// LS Electric XG5000 project: 신호등
// PLC LSPLC

PROGRAM NewProgram (task: 스캔 프로그램)

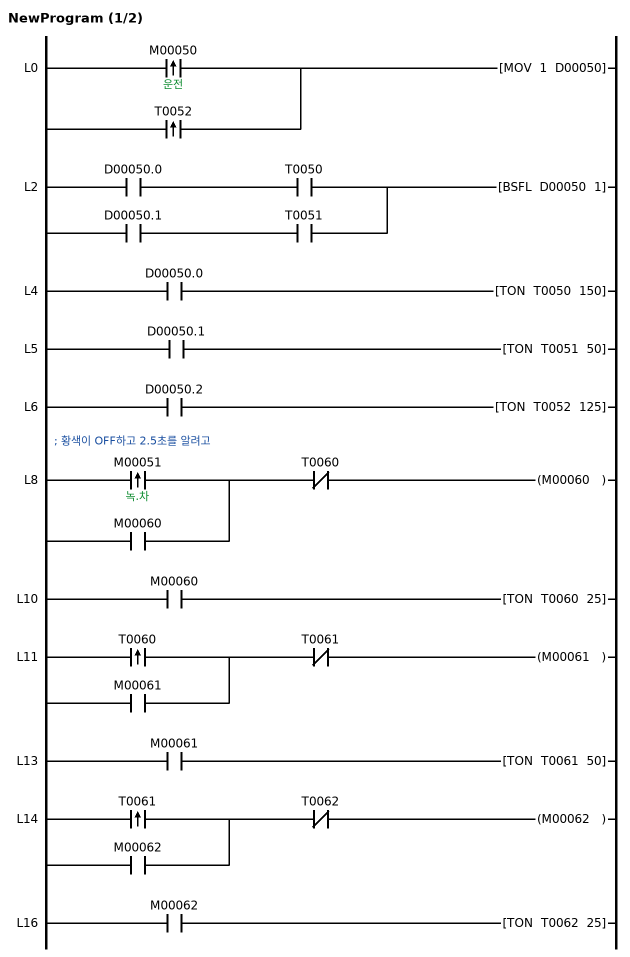
; L0
LOADP     M00050	// 운전
ORP       T0052
MOV       1 D00050
; L2
LOAD      D00050.0
AND       T0050
LOAD      D00050.1
AND       T0051
OR LOAD
BSFL      D00050 1
; L4
LOAD      D00050.0
TON       T0050 150
; L5
LOAD      D00050.1
TON       T0051 50
; L6
LOAD      D00050.2
TON       T0052 125
// 황색이 OFF하고 2.5초를 알려고
; L8
LOADP     M00051	// 녹.차
OR        M00060
AND NOT   T0060
OUT       M00060
; L10
LOAD      M00060
TON       T0060 25
; L11
LOADP     T0060
OR        M00061
AND NOT   T0061
OUT       M00061
; L13
LOAD      M00061
TON       T0061 50
; L14
LOADP     T0061
OR        M00062
AND NOT   T0062
OUT       M00062
; L16
LOAD      M00062
TON       T0062 25

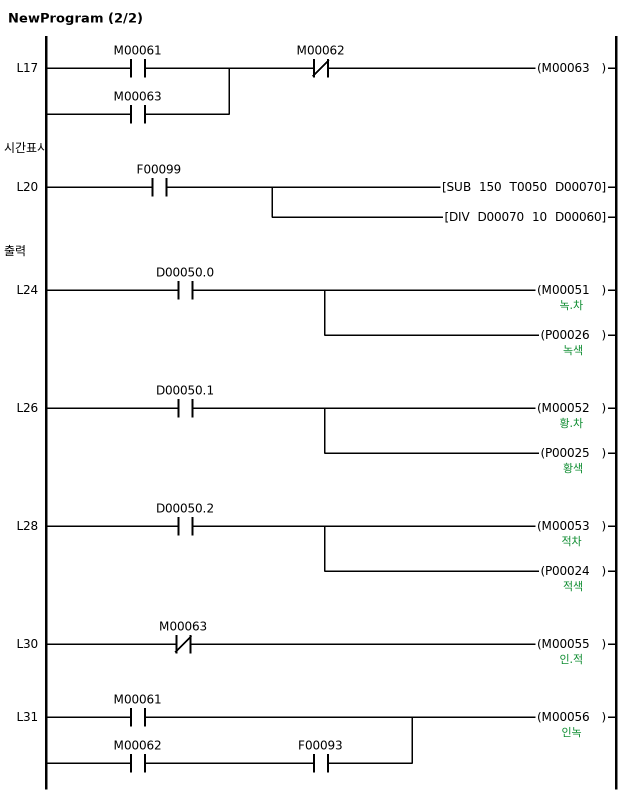
; L17
LOAD      M00061
OR        M00063
AND NOT   M00062
OUT       M00063
시간표시:
; L20
LOAD      F00099
SUB       150 T0050 D00070
DIV       D00070 10 D00060
출력:
; L24
LOAD      D00050.0
OUT       M00051	// 녹.차
OUT       P00026	// 녹색
; L26
LOAD      D00050.1
OUT       M00052	// 황.차
OUT       P00025	// 황색
; L28
LOAD      D00050.2
OUT       M00053	// 적차
OUT       P00024	// 적색
; L30
LOAD NOT  M00063
OUT       M00055	// 인.적
; L31
LOAD      M00061
LOAD      M00062
AND       F00093
OR LOAD
OUT       M00056	// 인녹

VARIABLES AND COMMENTS (devices not used above)
D00001	WORD	인.녹시간
M00090	BIT	황카운트
T0011	BIT/WORD	인.점.시
T0010	BIT/WORD	인.녹.시
T0012	BIT/WORD	다시적시작
T0001	BIT/WORD	인녹시
T0003	BIT/WORD	인점시
T0002	BIT/WORD	적.차.시
T0000	BIT/WORD	차.녹on